FUNCTION F_TMO_RoughVRC_ILK : BOOL
VAR_INPUT
	i_stISG : ST_VG; //Gauge measuring inlet Pressure e.g Pirani
	i_stBSG : ST_VG; //Gauge measuring backing Pressure e.g Pirani
	
END_VAR
VAR

	rInletPressureSP : REAL := 1E-03;
	rBackingPressureSP : REAL := 1E-03;
END_VAR

(* This Function Block evaluates the ILK condition of the roughing valve *)
(* The logic allows roughing valve to open when both inlet and backing pressure below than the SP*)

F_TMO_RoughVRC_ILK := (i_stISG.xPRESS_OK AND i_stISG.rPRESS < rInletPressureSP)
						AND (i_stBSG.xPRESS_OK AND i_stBSG.rPRESS < rBackingPressureSP);

END_FUNCTION

(* stored: Version 1.1.0.1, ProductVersion 3.1.4022.18
   POU F_TMO_RoughVRC_ILK: Id {923fd527-01a5-4fc8-9fca-a16621757af1}, SpecialFunc None *)
